KUKA KRL program: Sps5.sub

&ACCESS RV
&PARAM TPVW_VERSION=8.3.18
DEF  SPS5 ( )
; FOLD ;%{H} %MKUKATPVW
;Init part of vw_usr_s
VW_USR_S (#USR_INIT_SUB5)

LOOP
;Freilaufende SPS
MAKROSUBMIT5()

WAIT FOR NOT $POWER_FAIL
ENDLOOP
END
;ENDFOLD
